// TIA Portal V19 export
FUNCTION "Route 406" : Void   // FC105, FBD
TITLE = Polygon Transfer Line - Production Sequence
{ S7_Optimized_Access := 'TRUE' }
// stored: AutoNumber false, SetENOAutomatically false
   VAR_TEMP
      device_fault : Bool;
      switch_fault : Bool;
      tmp : Bool;
      Step_on : Bool;
      Dev_Check : Bool;
      New_Msg : Bool;
      Route_Ready : Bool;   // Ready to Run
      PNIOnodeFault : Bool;
      StepTime : S5Time;
      TimerError : Int;
      scratch_DI : DInt;
      scratch_Real : Real;
      Message : Int;
      scratch_I : Int;
      tmpWord : Word;
      PNIODiag : Struct
         node_2 : Struct
            failed : Bool;
            moduleFault : Bool;
         END_STRUCT;
         node_3 : Struct
            failed : Bool;
            moduleFault : Bool;
         END_STRUCT;
         node_4 : Struct
            failed : Bool;
            moduleFault : Bool;
         END_STRUCT;
         node_5 : Struct
            failed : Bool;
            moduleFault : Bool;
         END_STRUCT;
         node_6 : Struct
            failed : Bool;
            moduleFault : Bool;
         END_STRUCT;
         node_7 : Struct
            failed : Bool;
            moduleFault : Bool;
         END_STRUCT;
         node_8 : Struct
            failed : Bool;
            moduleFault : Bool;
         END_STRUCT;
         node_9 : Struct
            failed : Bool;
            moduleFault : Bool;
         END_STRUCT;
         node_10 : Struct
            failed : Bool;
            moduleFault : Bool;
         END_STRUCT;
         node_11 : Struct
            failed : Bool;
            moduleFault : Bool;
            node_10 : Struct
               failed : Bool;
               moduleFault : Bool;
            END_STRUCT;
         END_STRUCT;
         node_12 : Struct
            failed : Bool;
            moduleFault : Bool;
         END_STRUCT;
      END_STRUCT;
      TV_above_zero : Bool;
      TV_equal_zero : Bool;
      PNIO_FaultActive : Bool;
   END_VAR
   VAR_TEMP   // added for the SCL form of the ladder/FBD networks
      _w1 : Bool;
   END_VAR
BEGIN

NETWORK
TITLE = PNIO 100 Node Faults
// PNIO Node 2
// PNIO Node 2
      A     "Module Diagnostic Result"."2_AL1103".ErrorValue.%X1;
      =     #PNIODiag.node_2.failed;
      A     "Module Diagnostic Result"."2_AL1103".ErrorValue.%X2;
      =     #PNIODiag.node_2.moduleFault;
// PNIO Node 3
      A     "Module Diagnostic Result"."3_AL1307".ErrorValue.%X1;
      =     #PNIODiag.node_3.failed;
      A     "Module Diagnostic Result"."3_AL1307".ErrorValue.%X2;
      =     #PNIODiag.node_3.moduleFault;
// PNIO Node 4
      A     "Module Diagnostic Result"."4_AL1307".ErrorValue.%X1;
      =     #PNIODiag.node_4.failed;
      A     "Module Diagnostic Result"."4_AL1307".ErrorValue.%X2;
      =     #PNIODiag.node_4.moduleFault;
// PNIO Node 5
      A     "Module Diagnostic Result"."5_AL1307".ErrorValue.%X1;
      =     #PNIODiag.node_5.failed;
      A     "Module Diagnostic Result"."5_AL1307".ErrorValue.%X2;
      =     #PNIODiag.node_5.moduleFault;
// PNIO Node 6
      A     "Module Diagnostic Result"."6_AL1307".ErrorValue.%X1;
      =     #PNIODiag.node_6.failed;
      A     "Module Diagnostic Result"."6_AL1307".ErrorValue.%X2;
      =     #PNIODiag.node_6.moduleFault;
// PNIO Node 7
      A     "Module Diagnostic Result"."7_AL1307".ErrorValue.%X1;
      =     #PNIODiag.node_7.failed;
      A     "Module Diagnostic Result"."7_AL1307".ErrorValue.%X2;
      =     #PNIODiag.node_7.moduleFault;
// PNIO Node 8
      A     "Module Diagnostic Result"."8_Promag300".ErrorValue.%X1;
      =     #PNIODiag.node_8.failed;
      A     "Module Diagnostic Result"."8_Promag300".ErrorValue.%X2;
      =     #PNIODiag.node_8.moduleFault;
// PNIO Node 9
      A     "Module Diagnostic Result"."9_SinaG120".ErrorValue.%X1;
      =     #PNIODiag.node_9.failed;
      A     "Module Diagnostic Result"."9_SinaG120".ErrorValue.%X2;
      =     #PNIODiag.node_9.moduleFault;
// PNIO Node 10
      A     "Module Diagnostic Result"."10_AL1307".ErrorValue.%X1;
      =     #PNIODiag.node_10.failed;
      A     "Module Diagnostic Result"."10_AL1307".ErrorValue.%X2;
      =     #PNIODiag.node_10.moduleFault;
// PNIO Node 11
      A     "Module Diagnostic Result"."11_PNCoup".ErrorValue.%X1;
      =     #PNIODiag.node_11.failed;
      A     "Module Diagnostic Result"."11_PNCoup".ErrorValue.%X2;
      =     #PNIODiag.node_11.moduleFault;
// PNIO Node 12
      A     "Module Diagnostic Result"."12_AL1307".ErrorValue.%X1;
      =     #PNIODiag.node_12.failed;
      A     "Module Diagnostic Result"."12_AL1307".ErrorValue.%X2;
      =     #PNIODiag.node_12.moduleFault;


NETWORK
TITLE = PNIO node fault
      O     #PNIODiag.node_2.failed;
      O     #PNIODiag.node_2.moduleFault;
      O     #PNIODiag.node_3.failed;
      O     #PNIODiag.node_3.moduleFault;
      O     #PNIODiag.node_4.failed;
      O     #PNIODiag.node_4.moduleFault;
      O     #PNIODiag.node_5.failed;
      O     #PNIODiag.node_5.moduleFault;
      O     #PNIODiag.node_6.failed;
      O     #PNIODiag.node_6.moduleFault;
      O     #PNIODiag.node_7.failed;
      O     #PNIODiag.node_7.moduleFault;
      O     #PNIODiag.node_8.failed;
      O     #PNIODiag.node_8.moduleFault;
      O     #PNIODiag.node_9.failed;
      O     #PNIODiag.node_9.moduleFault;
      O     #PNIODiag.node_10.failed;
      O     #PNIODiag.node_10.moduleFault;
      O     #PNIODiag.node_11.failed;
      O     #PNIODiag.node_11.moduleFault;
      O     #PNIODiag.node_12.failed;
      O     #PNIODiag.node_12.moduleFault;
      AN    "RTE_406_DB".HMI_CMD.PNIO_FaultOverride;
      =     #PNIOnodeFault;


NETWORK
TITLE = PNIO Override
      A     "RTE_406_DB".HMI.SEQUENCE_HELD;
      A     #PNIOnodeFault;
      AN(;
      L     "IO-LinkDevicesDB".AL2221_100_005_X06.DeviceStatus;
      L     0;
      >I;
      O     #PNIODiag.node_5.failed;
      );
      S     "RTE_406_DB".HMI_CMD.PNIO_FaultOverrideAvail;

      AN    "RTE_406_DB".HMI.RUNNING;
      R     "RTE_406_DB".HMI_CMD.PNIO_FaultOverrideAvail;
      R     "RTE_406_DB".HMI_CMD.PNIO_FaultOverride;

REGION Network 4: Device Faults
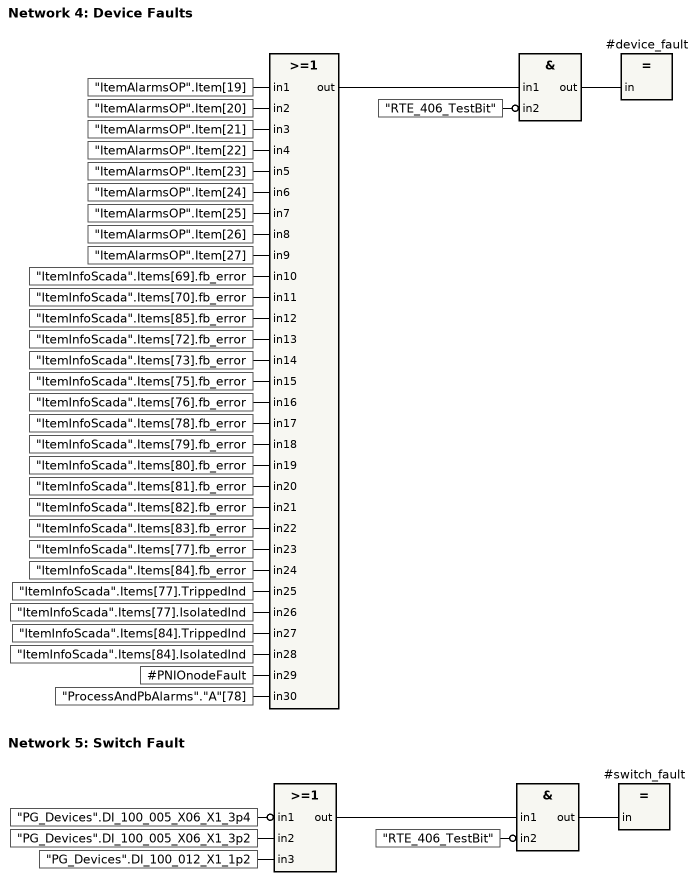
   #device_fault := ("ItemAlarmsOP".Item[19] OR "ItemAlarmsOP".Item[20] OR "ItemAlarmsOP".Item[21] OR "ItemAlarmsOP".Item[22] OR "ItemAlarmsOP".Item[23] OR "ItemAlarmsOP".Item[24] OR "ItemAlarmsOP".Item[25] OR "ItemAlarmsOP".Item[26] OR "ItemAlarmsOP".Item[27] OR "ItemInfoScada".Items[69].fb_error OR "ItemInfoScada".Items[70].fb_error OR "ItemInfoScada".Items[85].fb_error OR "ItemInfoScada".Items[72].fb_error OR "ItemInfoScada".Items[73].fb_error OR "ItemInfoScada".Items[75].fb_error OR "ItemInfoScada".Items[76].fb_error OR "ItemInfoScada".Items[78].fb_error OR "ItemInfoScada".Items[79].fb_error OR "ItemInfoScada".Items[80].fb_error OR "ItemInfoScada".Items[81].fb_error OR "ItemInfoScada".Items[82].fb_error OR "ItemInfoScada".Items[83].fb_error OR "ItemInfoScada".Items[77].fb_error OR "ItemInfoScada".Items[84].fb_error OR "ItemInfoScada".Items[77].TrippedInd OR "ItemInfoScada".Items[77].IsolatedInd OR "ItemInfoScada".Items[84].TrippedInd OR "ItemInfoScada".Items[84].IsolatedInd OR #PNIOnodeFault OR "ProcessAndPbAlarms"."A"[78]) AND NOT "RTE_406_TestBit";
END_REGION

REGION Network 5: Switch Fault
   #switch_fault := (NOT "PG_Devices".DI_100_005_X06_X1_3p4 OR "PG_Devices".DI_100_005_X06_X1_3p2 OR "PG_Devices".DI_100_012_X1_1p2) AND NOT "RTE_406_TestBit";
END_REGION

REGION Network 6: Set Devices in Auto
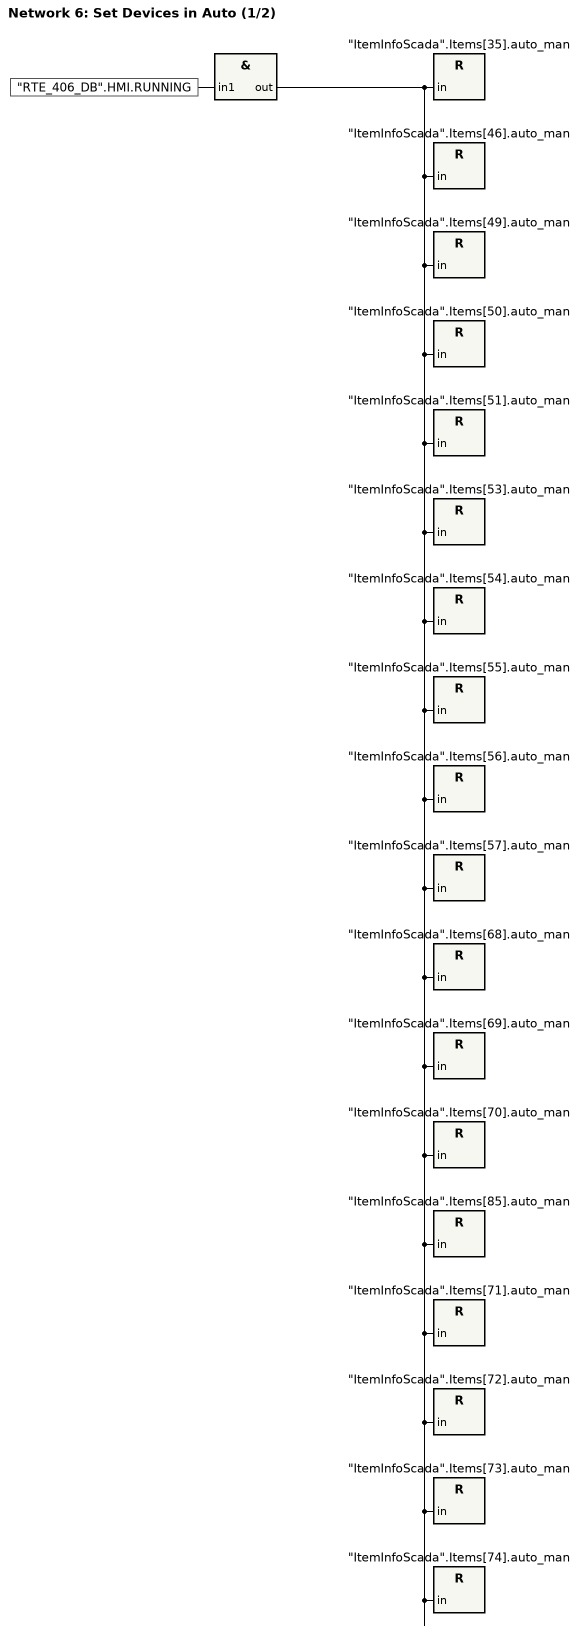
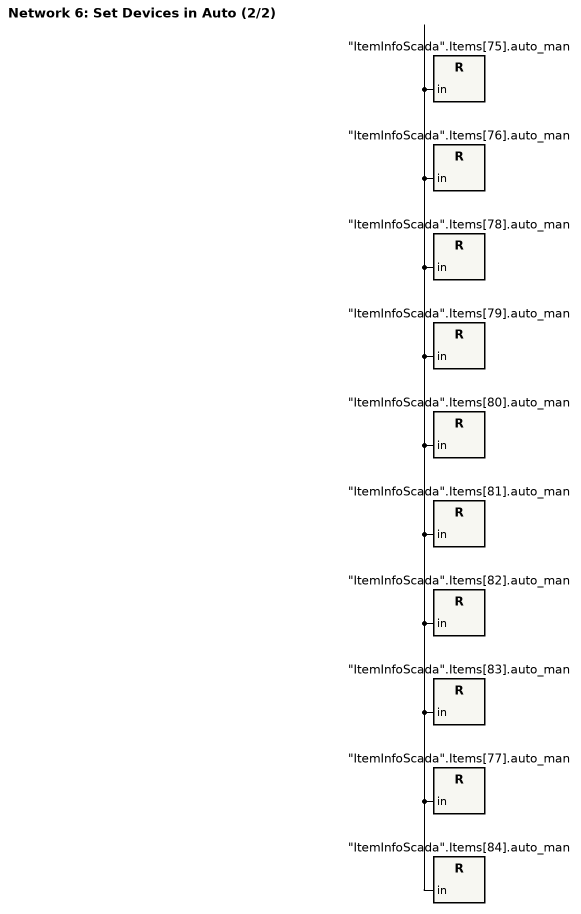
   IF "RTE_406_DB".HMI.RUNNING THEN
       "ItemInfoScada".Items[35].auto_man := FALSE;
       "ItemInfoScada".Items[46].auto_man := FALSE;
       "ItemInfoScada".Items[49].auto_man := FALSE;
       "ItemInfoScada".Items[50].auto_man := FALSE;
       "ItemInfoScada".Items[51].auto_man := FALSE;
       "ItemInfoScada".Items[53].auto_man := FALSE;
       "ItemInfoScada".Items[54].auto_man := FALSE;
       "ItemInfoScada".Items[55].auto_man := FALSE;
       "ItemInfoScada".Items[56].auto_man := FALSE;
       "ItemInfoScada".Items[57].auto_man := FALSE;
       "ItemInfoScada".Items[68].auto_man := FALSE;
       "ItemInfoScada".Items[69].auto_man := FALSE;
       "ItemInfoScada".Items[70].auto_man := FALSE;
       "ItemInfoScada".Items[85].auto_man := FALSE;
       "ItemInfoScada".Items[71].auto_man := FALSE;
       "ItemInfoScada".Items[72].auto_man := FALSE;
       "ItemInfoScada".Items[73].auto_man := FALSE;
       "ItemInfoScada".Items[74].auto_man := FALSE;
       "ItemInfoScada".Items[75].auto_man := FALSE;
       "ItemInfoScada".Items[76].auto_man := FALSE;
       "ItemInfoScada".Items[78].auto_man := FALSE;
       "ItemInfoScada".Items[79].auto_man := FALSE;
       "ItemInfoScada".Items[80].auto_man := FALSE;
       "ItemInfoScada".Items[81].auto_man := FALSE;
       "ItemInfoScada".Items[82].auto_man := FALSE;
       "ItemInfoScada".Items[83].auto_man := FALSE;
       "ItemInfoScada".Items[77].auto_man := FALSE;
       "ItemInfoScada".Items[84].auto_man := FALSE;
   END_IF;
END_REGION

REGION Network 7: Route Healthy
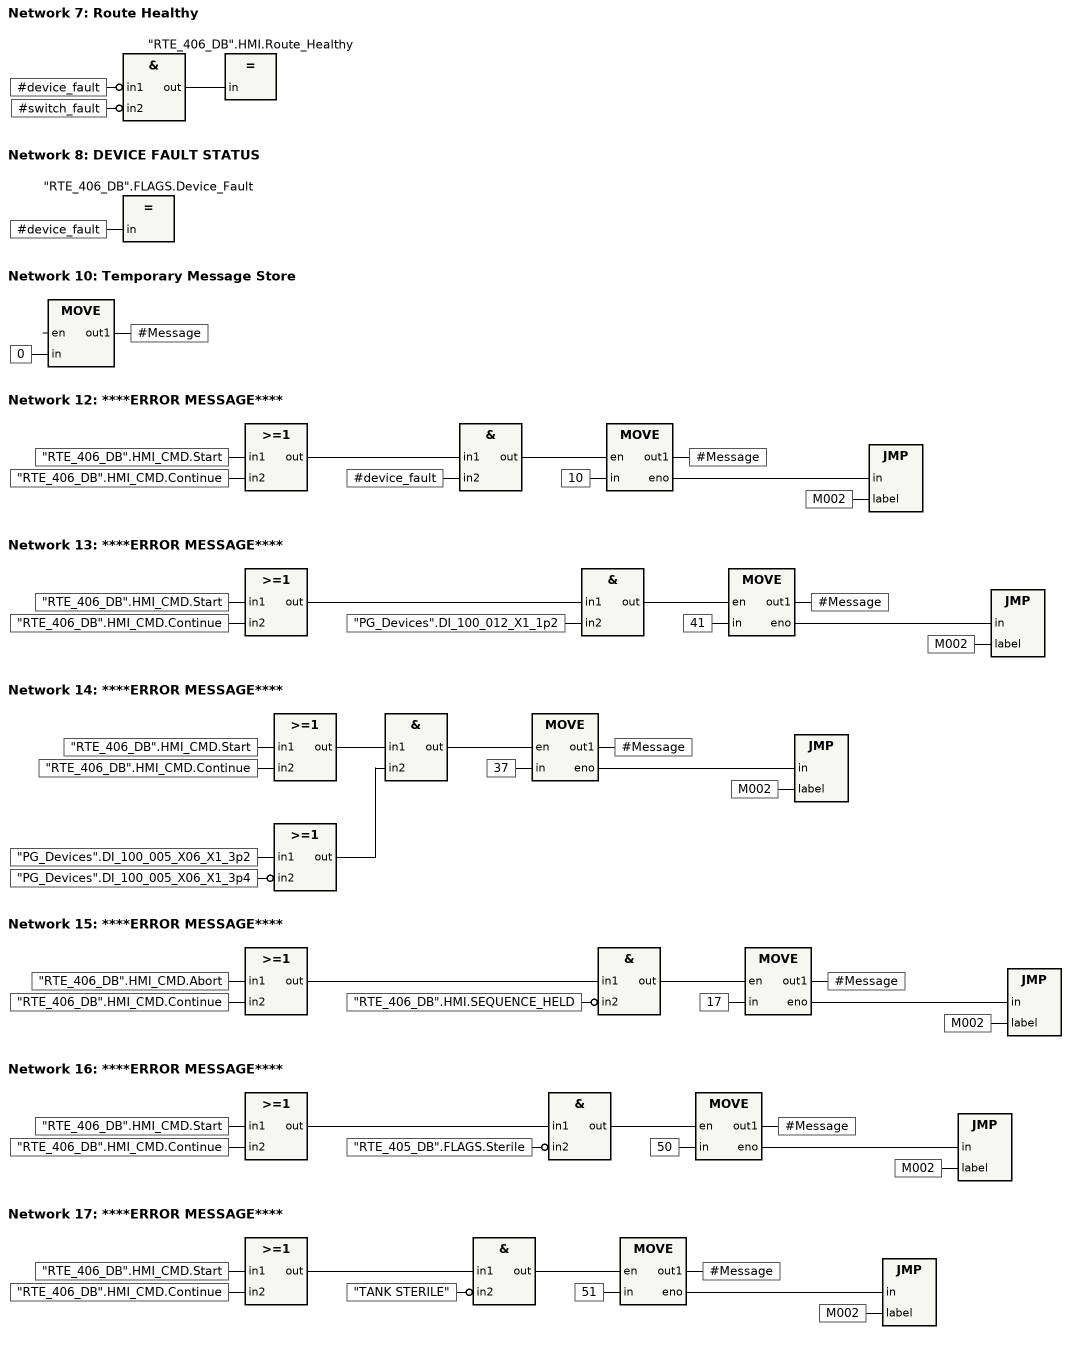
   "RTE_406_DB".HMI.Route_Healthy := NOT #device_fault AND NOT #switch_fault;
END_REGION

REGION Network 8: DEVICE FAULT STATUS
   "RTE_406_DB".FLAGS.Device_Fault := #device_fault;
END_REGION

NETWORK
TITLE = GENERAL FAULT STATUS
      O     #switch_fault;
      O     "RTE_406_DB".FLAGS.Device_Fault;
      A     "RTE_406_DB".HMI.RUNNING;
      =     "RTE_406_DB".HMI.FAULT;

REGION Network 10: Temporary Message Store
   // Clear down temporary message store.
   #Message := 0;
END_REGION

NETWORK
TITLE = Generate Sequence Start Command
// The sequence is initiated via the interface signals ..afl
      A     "RTE_406_DB".HMI_CMD.Start;
      AN    "RTE_406_DB".HMI.RUNNING;
      A     "RTE_406_DB".HMI.Route_Healthy;
      =     "RTE_406_DB".FLAGS.Sequence_Start;

      AN    "RTE_406_DB".HMI.RUNNING;
      A     "RTE_406_DB".HMI.Route_Healthy;
      =     "RTE_406_DB".HMI_CMD.Start_Available;


REGION Network 12: ****ERROR MESSAGE****
   // Message 10 - Device Fault
   // ENO of a box is taken as its EN; it also drops when the box reports an error
   #_w1 := ("RTE_406_DB".HMI_CMD.Start OR "RTE_406_DB".HMI_CMD.Continue) AND #device_fault;
   IF #_w1 THEN
       #Message := 10;
       GOTO M002;
   END_IF;
END_REGION

REGION Network 13: ****ERROR MESSAGE****
   // Message 41 - Forward Control Stop activated
   // ENO of a box is taken as its EN; it also drops when the box reports an error
   #_w1 := ("RTE_406_DB".HMI_CMD.Start OR "RTE_406_DB".HMI_CMD.Continue) AND "PG_Devices".DI_100_012_X1_1p2;
   IF #_w1 THEN
       #Message := 41;
       GOTO M002;
   END_IF;
END_REGION

REGION Network 14: ****ERROR MESSAGE****
   // Message 37 - Swingbend out of position
   // ENO of a box is taken as its EN; it also drops when the box reports an error
   #_w1 := ("RTE_406_DB".HMI_CMD.Start OR "RTE_406_DB".HMI_CMD.Continue) AND ("PG_Devices".DI_100_005_X06_X1_3p2 OR NOT "PG_Devices".DI_100_005_X06_X1_3p4);
   IF #_w1 THEN
       #Message := 37;
       GOTO M002;
   END_IF;
END_REGION

REGION Network 15: ****ERROR MESSAGE****
   // Message 17 - Sequence Not Held
   // To abort or continue the clean it must have already been held.
   // ENO of a box is taken as its EN; it also drops when the box reports an error
   #_w1 := ("RTE_406_DB".HMI_CMD.Abort OR "RTE_406_DB".HMI_CMD.Continue) AND NOT "RTE_406_DB".HMI.SEQUENCE_HELD;
   IF #_w1 THEN
       #Message := 17;
       GOTO M002;
   END_IF;
END_REGION

REGION Network 16: ****ERROR MESSAGE****
   // Message 50 - Line not Sterile
   // ENO of a box is taken as its EN; it also drops when the box reports an error
   #_w1 := ("RTE_406_DB".HMI_CMD.Start OR "RTE_406_DB".HMI_CMD.Continue) AND NOT "RTE_405_DB".FLAGS.Sterile;
   IF #_w1 THEN
       #Message := 50;
       GOTO M002;
   END_IF;
END_REGION

REGION Network 17: ****ERROR MESSAGE****
   // Message 51 - AHV Not Sterile
   // ENO of a box is taken as its EN; it also drops when the box reports an error
   #_w1 := ("RTE_406_DB".HMI_CMD.Start OR "RTE_406_DB".HMI_CMD.Continue) AND NOT "TANK STERILE";
   IF #_w1 THEN
       #Message := 51;
       GOTO M002;
   END_IF;
END_REGION

REGION Network 18: ****ERROR MESSAGE****
   // Message 28 - Filler Not Sterile
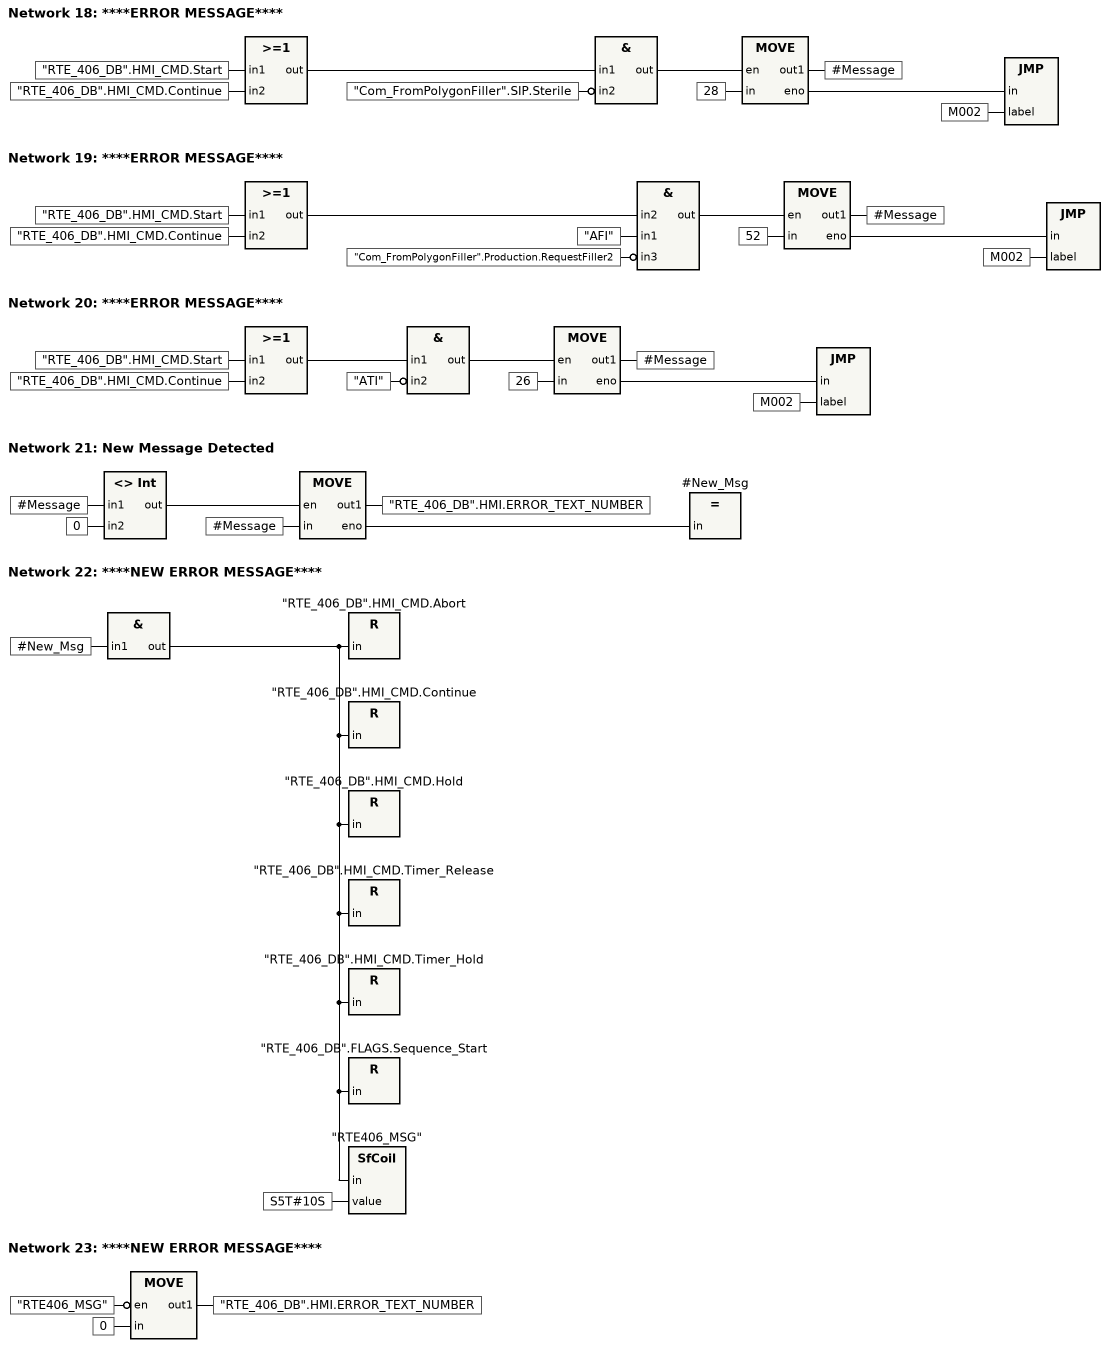
   // ENO of a box is taken as its EN; it also drops when the box reports an error
   #_w1 := ("RTE_406_DB".HMI_CMD.Start OR "RTE_406_DB".HMI_CMD.Continue) AND NOT "Com_FromPolygonFiller".SIP.Sterile;
   IF #_w1 THEN
       #Message := 28;
       GOTO M002;
   END_IF;
END_REGION

REGION Network 19: ****ERROR MESSAGE****
   // Message 52 - No Product Request From Filler
   // ENO of a box is taken as its EN; it also drops when the box reports an error
   #_w1 := ("RTE_406_DB".HMI_CMD.Start OR "RTE_406_DB".HMI_CMD.Continue) AND "AFI" AND NOT "Com_FromPolygonFiller".Production.RequestFiller2;
   IF #_w1 THEN
       #Message := 52;
       GOTO M002;
   END_IF;
END_REGION

REGION Network 20: ****ERROR MESSAGE****
   // Message xx - Tank low level for production start
   // Check text msg number
   // ENO of a box is taken as its EN; it also drops when the box reports an error
   #_w1 := ("RTE_406_DB".HMI_CMD.Start OR "RTE_406_DB".HMI_CMD.Continue) AND NOT "ATI";
   IF #_w1 THEN
       #Message := 26;
       GOTO M002;
   END_IF;
END_REGION

REGION Network 21: New Message Detected
   // ENO of a box is taken as its EN; it also drops when the box reports an error
   M002:
   #_w1 := #Message <> 0;
   IF #_w1 THEN "RTE_406_DB".HMI.ERROR_TEXT_NUMBER := #Message; END_IF;
   #New_Msg := #_w1;
END_REGION

REGION Network 22: ****NEW ERROR MESSAGE****
   // Reset all CIP commands except START.
   // On a new non-zero error message being displayed reset all commands from SCADA 
   // so they take no action. Also, start a delay off timer to cancel display of the 
   // error message.
   // no SCL statement known for SfCoil: written as a call
   IF #New_Msg THEN
       "RTE_406_DB".HMI_CMD.Abort := FALSE;
       "RTE_406_DB".HMI_CMD.Continue := FALSE;
       "RTE_406_DB".HMI_CMD.Hold := FALSE;
       "RTE_406_DB".HMI_CMD.Timer_Release := FALSE;
       "RTE_406_DB".HMI_CMD.Timer_Hold := FALSE;
       "RTE_406_DB".FLAGS.Sequence_Start := FALSE;
   END_IF;
   SfCoil(in := #New_Msg, value := S5T#10S, operand := "RTE406_MSG");
END_REGION

REGION Network 23: ****NEW ERROR MESSAGE****
   // Error message display cancel.
   IF NOT "RTE406_MSG" THEN "RTE_406_DB".HMI.ERROR_TEXT_NUMBER := 0; END_IF;
END_REGION

REGION Network 24: ROUTE RUNNING
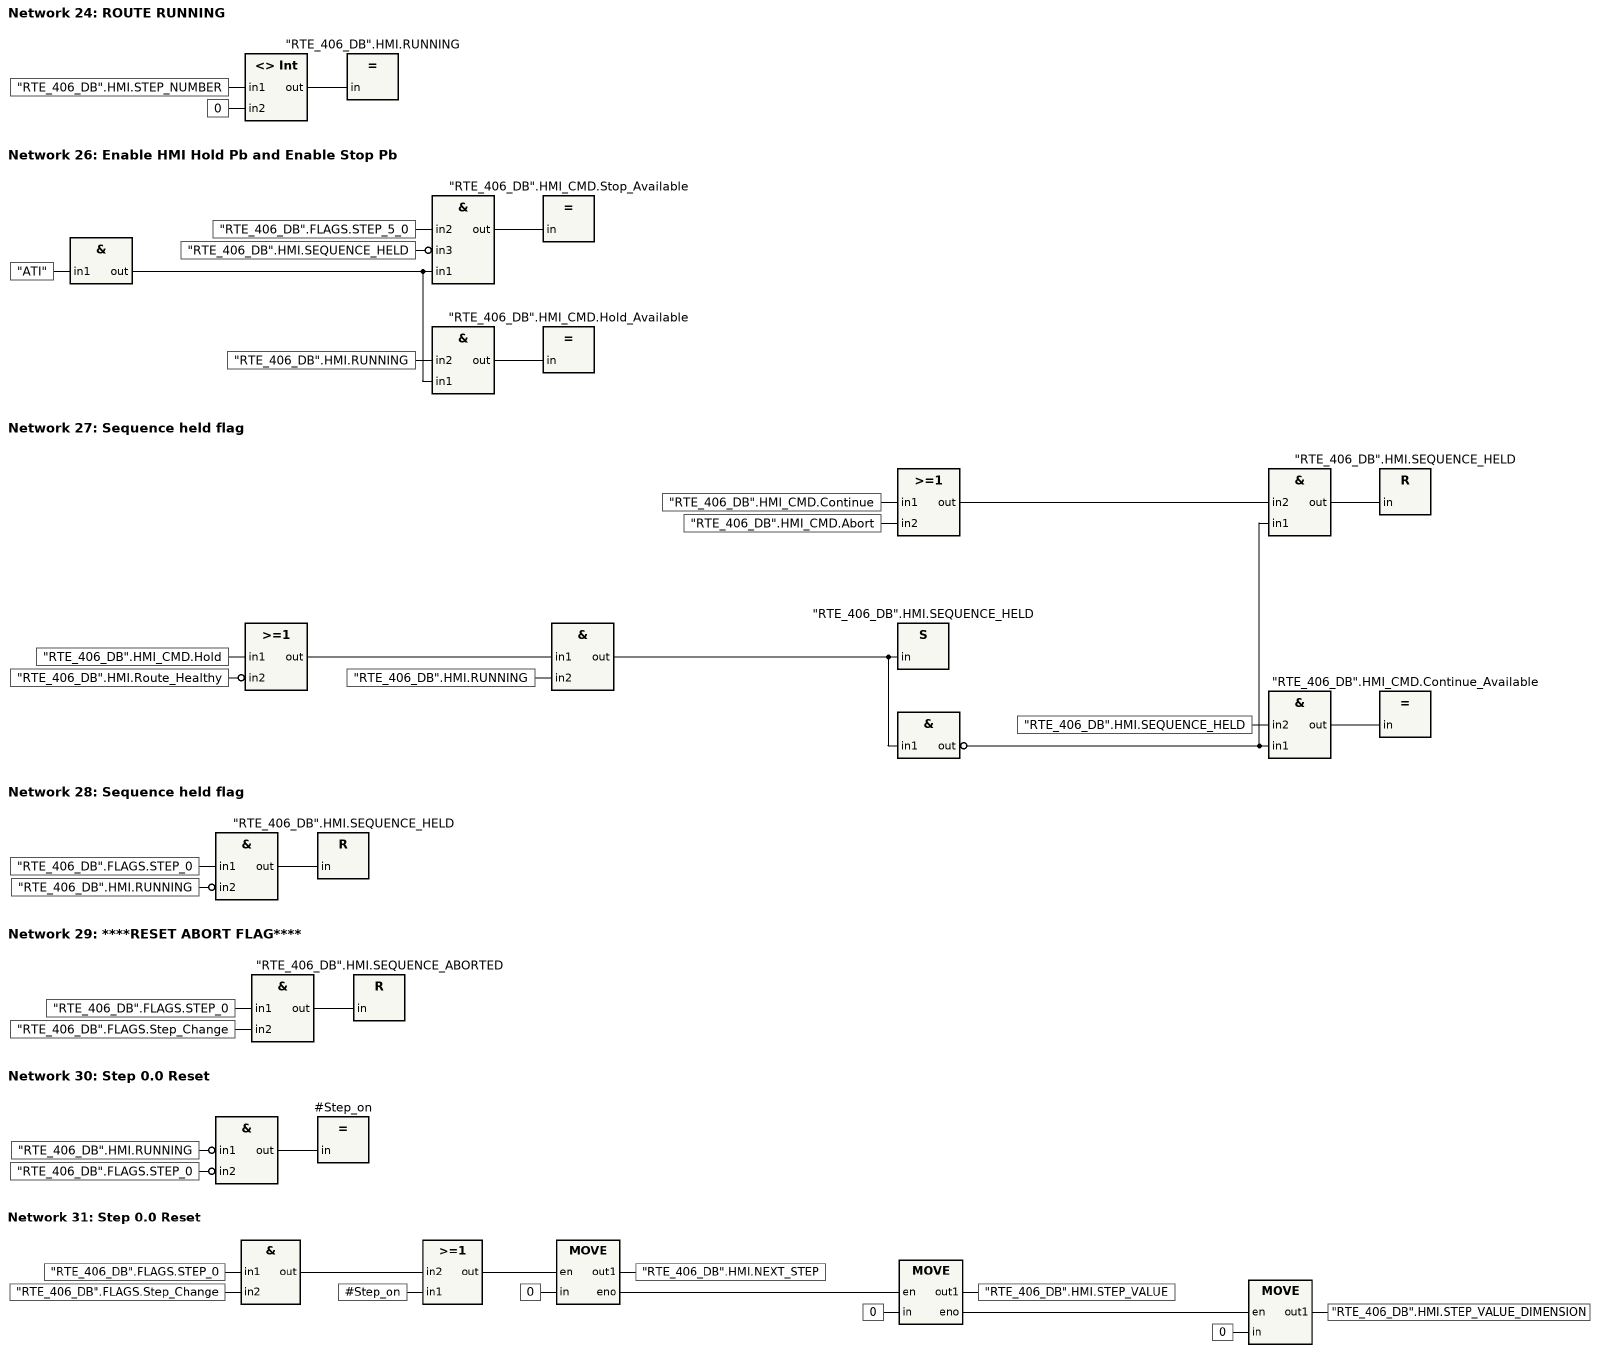
   "RTE_406_DB".HMI.RUNNING := "RTE_406_DB".HMI.STEP_NUMBER <> 0;
END_REGION

NETWORK
TITLE = ****SEQ ABORT****
      A     "RTE_406_DB".HMI_CMD.Abort;
      A     "RTE_406_DB".HMI.SEQUENCE_HELD;
      S     "RTE_406_DB".HMI.SEQUENCE_ABORTED;

      A     "RTE_406_DB".HMI.SEQUENCE_HELD;
      =     "RTE_406_DB".HMI_CMD.Abort_Available;

REGION Network 26: Enable HMI Hold Pb and Enable Stop Pb
   "RTE_406_DB".HMI_CMD.Hold_Available := "RTE_406_DB".HMI.RUNNING AND "ATI";
   "RTE_406_DB".HMI_CMD.Stop_Available := "RTE_406_DB".FLAGS.STEP_5_0 AND NOT "RTE_406_DB".HMI.SEQUENCE_HELD AND "ATI";
END_REGION

REGION Network 27: Sequence held flag
   // Set sequence hold if sequence is running and a hold fault condition is detected 
   // or a sequence hold command is received from SCADA.
   // 
   // When a validated CONTINUE command is received from SCADA and all fault 
   // conditions are cleared then reset sequence hold.
   #_w1 := ("RTE_406_DB".HMI_CMD.Hold OR NOT "RTE_406_DB".HMI.Route_Healthy) AND "RTE_406_DB".HMI.RUNNING;
   IF #_w1 THEN "RTE_406_DB".HMI.SEQUENCE_HELD := TRUE; END_IF;
   IF ("RTE_406_DB".HMI_CMD.Continue OR "RTE_406_DB".HMI_CMD.Abort) AND NOT #_w1 THEN
       "RTE_406_DB".HMI.SEQUENCE_HELD := FALSE;
   END_IF;
   "RTE_406_DB".HMI_CMD.Continue_Available := "RTE_406_DB".HMI.SEQUENCE_HELD AND NOT #_w1;
END_REGION

REGION Network 28: Sequence held flag
   // Reset when circuit not running i.e after an abort.
   IF "RTE_406_DB".FLAGS.STEP_0 AND NOT "RTE_406_DB".HMI.RUNNING THEN
       "RTE_406_DB".HMI.SEQUENCE_HELD := FALSE;
   END_IF;
END_REGION

REGION Network 29: ****RESET ABORT FLAG****
   IF "RTE_406_DB".FLAGS.STEP_0 AND "RTE_406_DB".FLAGS.Step_Change THEN
       "RTE_406_DB".HMI.SEQUENCE_ABORTED := FALSE;
   END_IF;
END_REGION

REGION Network 30: Step 0.0 Reset
   #Step_on := NOT "RTE_406_DB".HMI.RUNNING AND NOT "RTE_406_DB".FLAGS.STEP_0;
END_REGION

REGION Network 31: Step 0.0 Reset
   // Reset sequnece to step 0 and clear down step value and dimension words.
   // ENO of a box is taken as its EN; it also drops when the box reports an error
   IF ("RTE_406_DB".FLAGS.STEP_0 AND "RTE_406_DB".FLAGS.Step_Change) OR #Step_on THEN
       "RTE_406_DB".HMI.NEXT_STEP := 0;
       "RTE_406_DB".HMI.STEP_VALUE := 0;
       "RTE_406_DB".HMI.STEP_VALUE_DIMENSION := 0;
   END_IF;
END_REGION

REGION Network 32: Move to Step 0.5
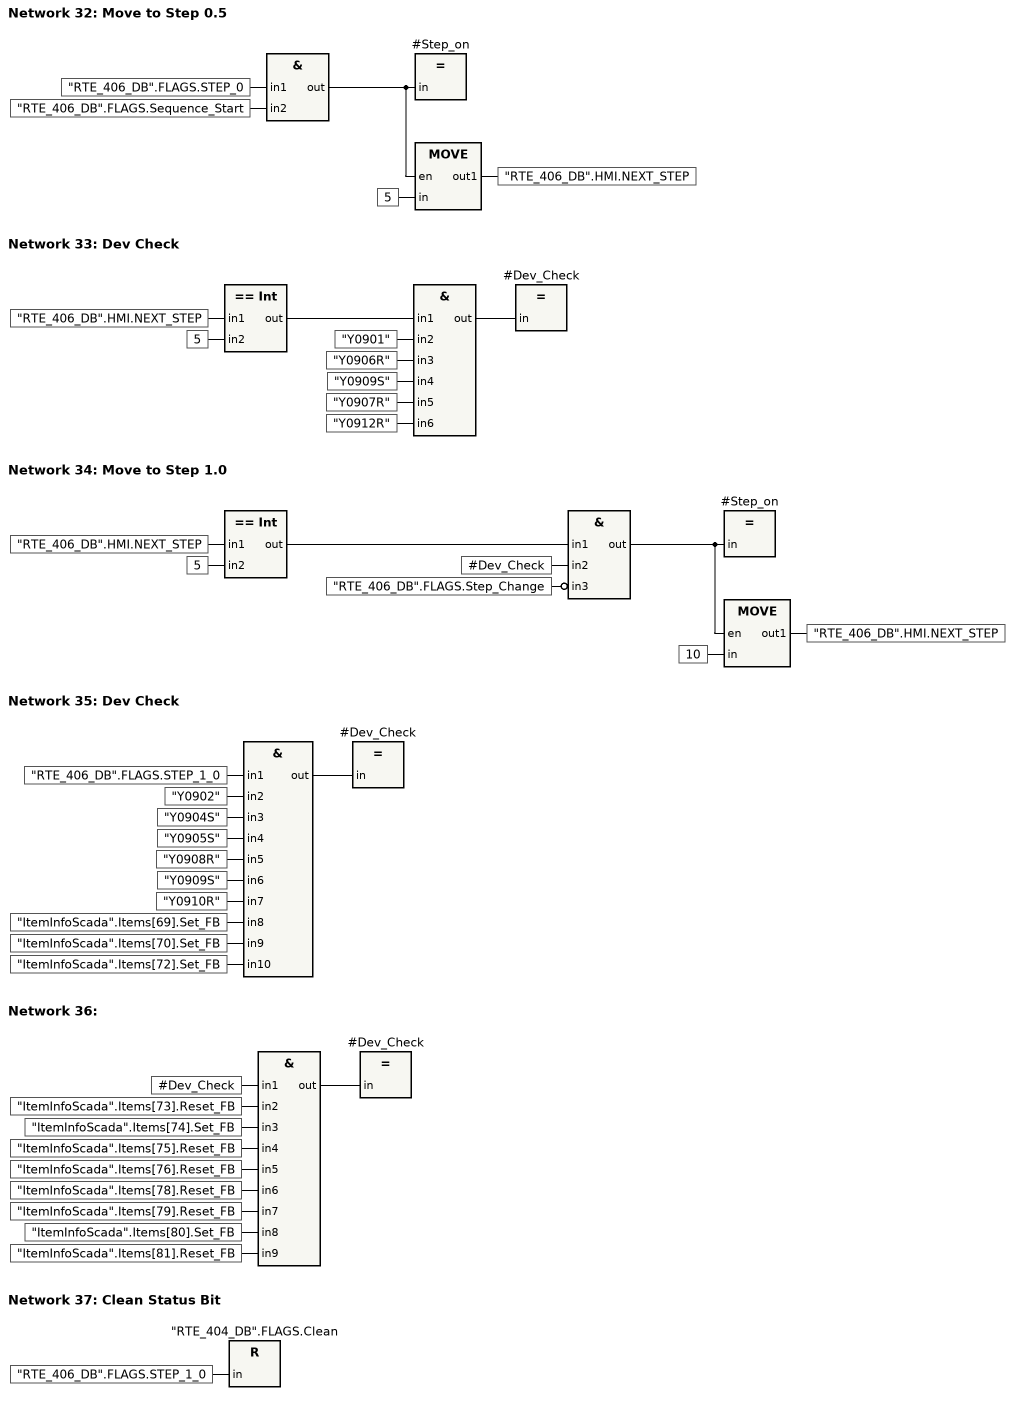
   #Step_on := "RTE_406_DB".FLAGS.STEP_0 AND "RTE_406_DB".FLAGS.Sequence_Start;
   IF #Step_on THEN "RTE_406_DB".HMI.NEXT_STEP := 5; END_IF;
END_REGION

REGION Network 33: Dev Check
   // Dev Check following Route valves Open - 09.10, 09.08, 09.45, 10.21, 10.23, 10.25
   // and following Route Valves closed - 09.09, 09.05, 10.24
   #Dev_Check := ("RTE_406_DB".HMI.NEXT_STEP = 5) AND "Y0901" AND "Y0906R" AND "Y0909S" AND "Y0907R" AND "Y0912R";
END_REGION

REGION Network 34: Move to Step 1.0
   #Step_on := ("RTE_406_DB".HMI.NEXT_STEP = 5) AND #Dev_Check AND NOT "RTE_406_DB".FLAGS.Step_Change;
   IF #Step_on THEN "RTE_406_DB".HMI.NEXT_STEP := 10; END_IF;
END_REGION

REGION Network 35: Dev Check
   // Dev Check following Route valves Open - 09.10, 09.08, 09.45, 10.21, 10.23, 10.25
   // and following Route Valves closed - 09.09, 09.05, 10.24
   #Dev_Check := "RTE_406_DB".FLAGS.STEP_1_0 AND "Y0902" AND "Y0904S" AND "Y0905S" AND "Y0908R" AND "Y0909S" AND "Y0910R" AND "ItemInfoScada".Items[69].Set_FB AND "ItemInfoScada".Items[70].Set_FB AND "ItemInfoScada".Items[72].Set_FB;
END_REGION

REGION Network 36
   #Dev_Check := #Dev_Check AND "ItemInfoScada".Items[73].Reset_FB AND "ItemInfoScada".Items[74].Set_FB AND "ItemInfoScada".Items[75].Reset_FB AND "ItemInfoScada".Items[76].Reset_FB AND "ItemInfoScada".Items[78].Reset_FB AND "ItemInfoScada".Items[79].Reset_FB AND "ItemInfoScada".Items[80].Set_FB AND "ItemInfoScada".Items[81].Reset_FB;
END_REGION

REGION Network 37: Clean Status Bit
   IF "RTE_406_DB".FLAGS.STEP_1_0 THEN "RTE_404_DB".FLAGS.Clean := FALSE; END_IF;
END_REGION

REGION Network 38: Move to Step 2.0
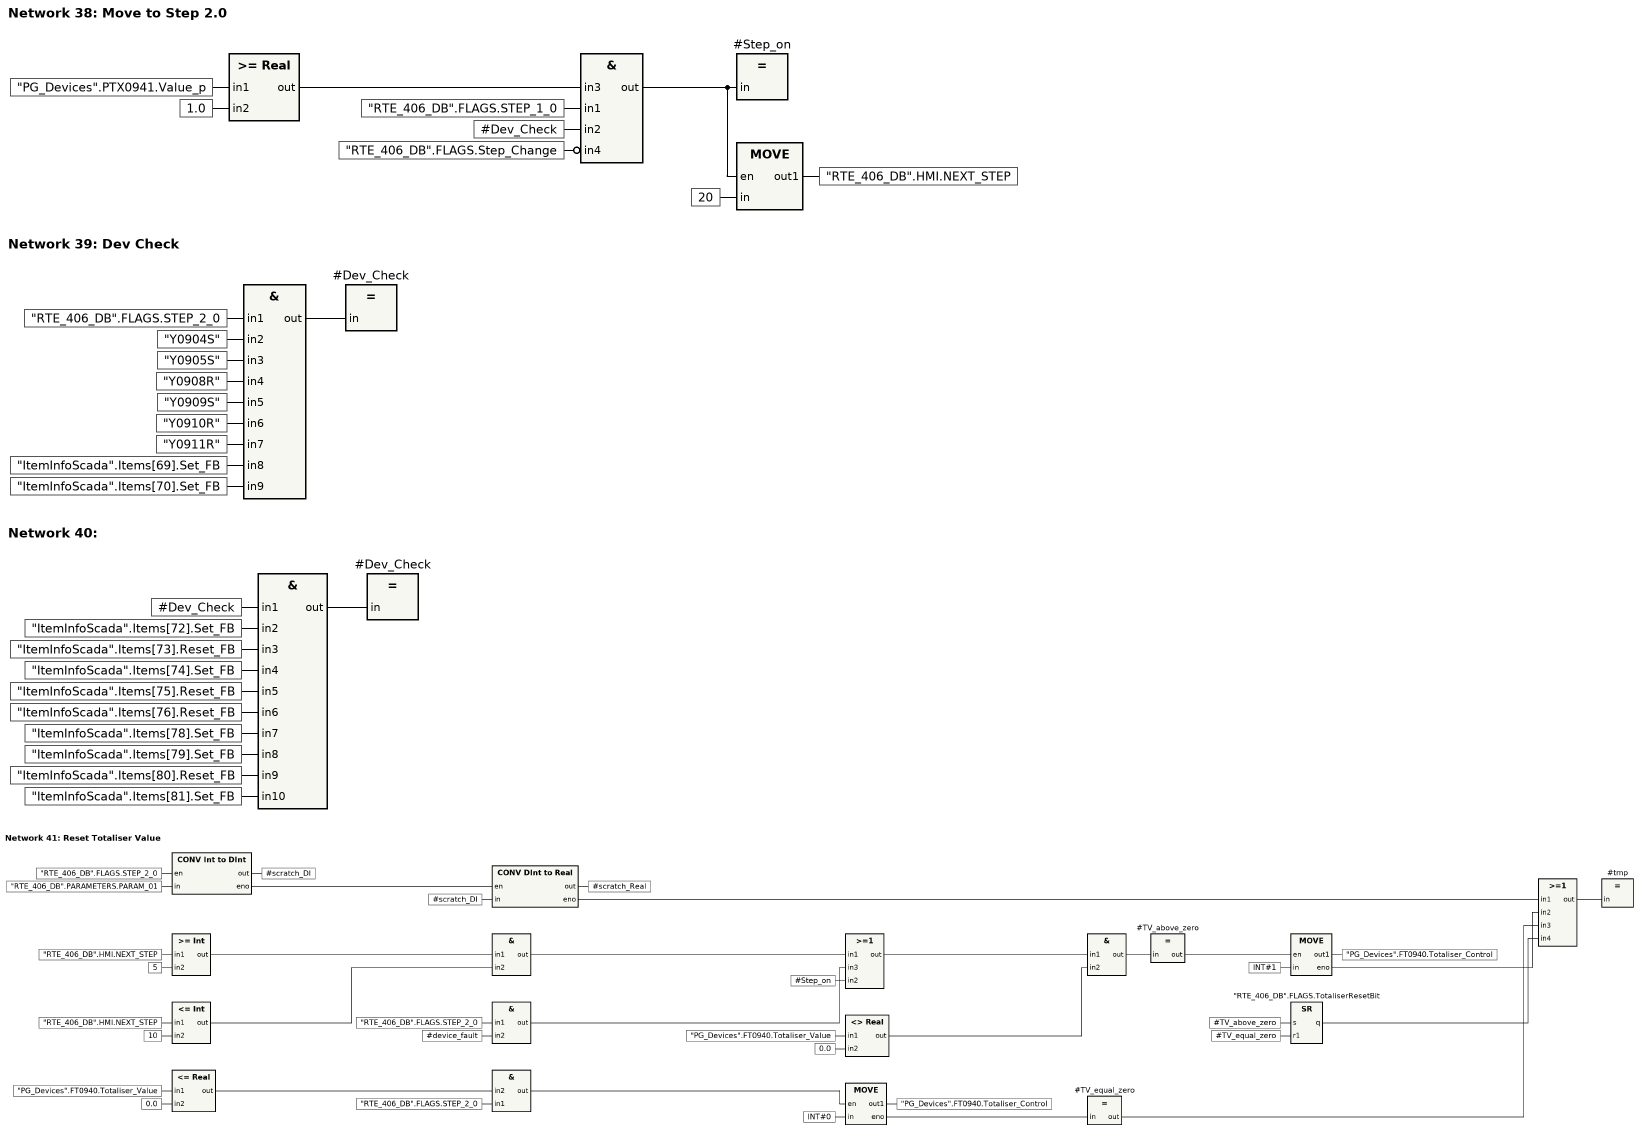
   #Step_on := ("PG_Devices".PTX0941.Value_p >= 1.0) AND "RTE_406_DB".FLAGS.STEP_1_0 AND #Dev_Check AND NOT "RTE_406_DB".FLAGS.Step_Change;
   IF #Step_on THEN "RTE_406_DB".HMI.NEXT_STEP := 20; END_IF;
END_REGION

REGION Network 39: Dev Check
   // Dev Check following Route valves Open - 09.10, 09.08, 09.45, 10.21, 10.23, 10.25
   // and following Route Valves closed - 09.09, 09.05, 10.24
   #Dev_Check := "RTE_406_DB".FLAGS.STEP_2_0 AND "Y0904S" AND "Y0905S" AND "Y0908R" AND "Y0909S" AND "Y0910R" AND "Y0911R" AND "ItemInfoScada".Items[69].Set_FB AND "ItemInfoScada".Items[70].Set_FB;
END_REGION

REGION Network 40
   #Dev_Check := #Dev_Check AND "ItemInfoScada".Items[72].Set_FB AND "ItemInfoScada".Items[73].Reset_FB AND "ItemInfoScada".Items[74].Set_FB AND "ItemInfoScada".Items[75].Reset_FB AND "ItemInfoScada".Items[76].Reset_FB AND "ItemInfoScada".Items[78].Set_FB AND "ItemInfoScada".Items[79].Set_FB AND "ItemInfoScada".Items[80].Reset_FB AND "ItemInfoScada".Items[81].Set_FB;
END_REGION

REGION Network 41: Reset Totaliser Value
   // Totaliser Control
   // 0 = Totalise
   // 3 = Reset + Totalise
   // ENO of a box is taken as its EN; it also drops when the box reports an error
   IF "RTE_406_DB".FLAGS.STEP_2_0 THEN
       #scratch_DI := INT_TO_DINT("RTE_406_DB".PARAMETERS.PARAM_01);
       #scratch_Real := DINT_TO_REAL(#scratch_DI);
   END_IF;
   #TV_above_zero := ((("RTE_406_DB".HMI.NEXT_STEP >= 5) AND ("RTE_406_DB".HMI.NEXT_STEP <= 10)) OR ("RTE_406_DB".FLAGS.STEP_2_0 AND #device_fault) OR #Step_on) AND ("PG_Devices".FT0940.Totaliser_Value <> 0.0);
   IF #TV_above_zero THEN "PG_Devices".FT0940.Totaliser_Control := INT#1; END_IF;
   #_w1 := ("PG_Devices".FT0940.Totaliser_Value <= 0.0) AND "RTE_406_DB".FLAGS.STEP_2_0;
   IF #_w1 THEN "PG_Devices".FT0940.Totaliser_Control := INT#0; END_IF;
   #TV_equal_zero := #_w1;
   IF #TV_above_zero THEN
       "RTE_406_DB".FLAGS.TotaliserResetBit := TRUE;   // SR flip-flop
   END_IF;
   IF #TV_equal_zero THEN "RTE_406_DB".FLAGS.TotaliserResetBit := FALSE; END_IF;
   #tmp := "RTE_406_DB".FLAGS.STEP_2_0 OR #TV_above_zero OR #_w1 OR "RTE_406_DB".FLAGS.TotaliserResetBit;
END_REGION

REGION Network 42: Move to Step 3.0
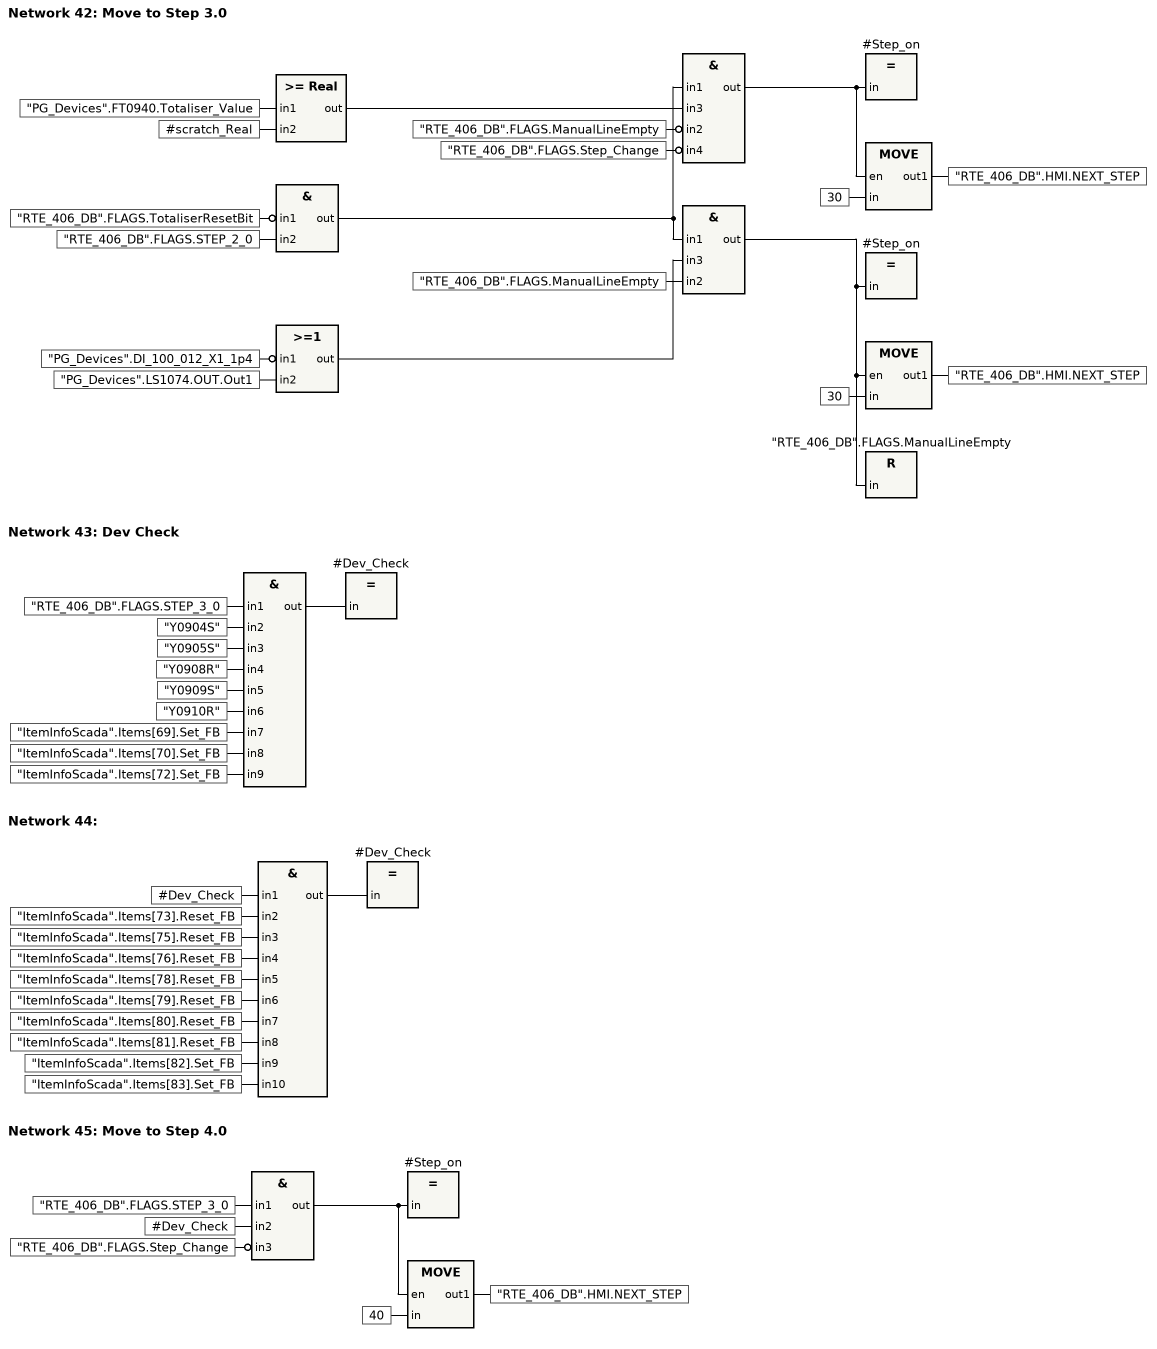
   #_w1 := NOT "RTE_406_DB".FLAGS.TotaliserResetBit AND "RTE_406_DB".FLAGS.STEP_2_0;
   #Step_on := #_w1 AND ("PG_Devices".FT0940.Totaliser_Value >= #scratch_Real) AND NOT "RTE_406_DB".FLAGS.ManualLineEmpty AND NOT "RTE_406_DB".FLAGS.Step_Change;
   IF #Step_on THEN "RTE_406_DB".HMI.NEXT_STEP := 30; END_IF;
   #Step_on := #_w1 AND (NOT "PG_Devices".DI_100_012_X1_1p4 OR "PG_Devices".LS1074.OUT.Out1) AND "RTE_406_DB".FLAGS.ManualLineEmpty;
   IF #Step_on THEN
       "RTE_406_DB".HMI.NEXT_STEP := 30;
       "RTE_406_DB".FLAGS.ManualLineEmpty := FALSE;
   END_IF;
END_REGION

REGION Network 43: Dev Check
   // Dev Check following Route valves Open - 09.10, 09.08, 09.45, 10.21, 10.23, 10.25
   // and following Route Valves closed - 09.09, 09.05, 10.24
   #Dev_Check := "RTE_406_DB".FLAGS.STEP_3_0 AND "Y0904S" AND "Y0905S" AND "Y0908R" AND "Y0909S" AND "Y0910R" AND "ItemInfoScada".Items[69].Set_FB AND "ItemInfoScada".Items[70].Set_FB AND "ItemInfoScada".Items[72].Set_FB;
END_REGION

REGION Network 44
   #Dev_Check := #Dev_Check AND "ItemInfoScada".Items[73].Reset_FB AND "ItemInfoScada".Items[75].Reset_FB AND "ItemInfoScada".Items[76].Reset_FB AND "ItemInfoScada".Items[78].Reset_FB AND "ItemInfoScada".Items[79].Reset_FB AND "ItemInfoScada".Items[80].Reset_FB AND "ItemInfoScada".Items[81].Reset_FB AND "ItemInfoScada".Items[82].Set_FB AND "ItemInfoScada".Items[83].Set_FB;
END_REGION

REGION Network 45: Move to Step 4.0
   #Step_on := "RTE_406_DB".FLAGS.STEP_3_0 AND #Dev_Check AND NOT "RTE_406_DB".FLAGS.Step_Change;
   IF #Step_on THEN "RTE_406_DB".HMI.NEXT_STEP := 40; END_IF;
END_REGION

REGION Network 46: Initialise Step Parameters
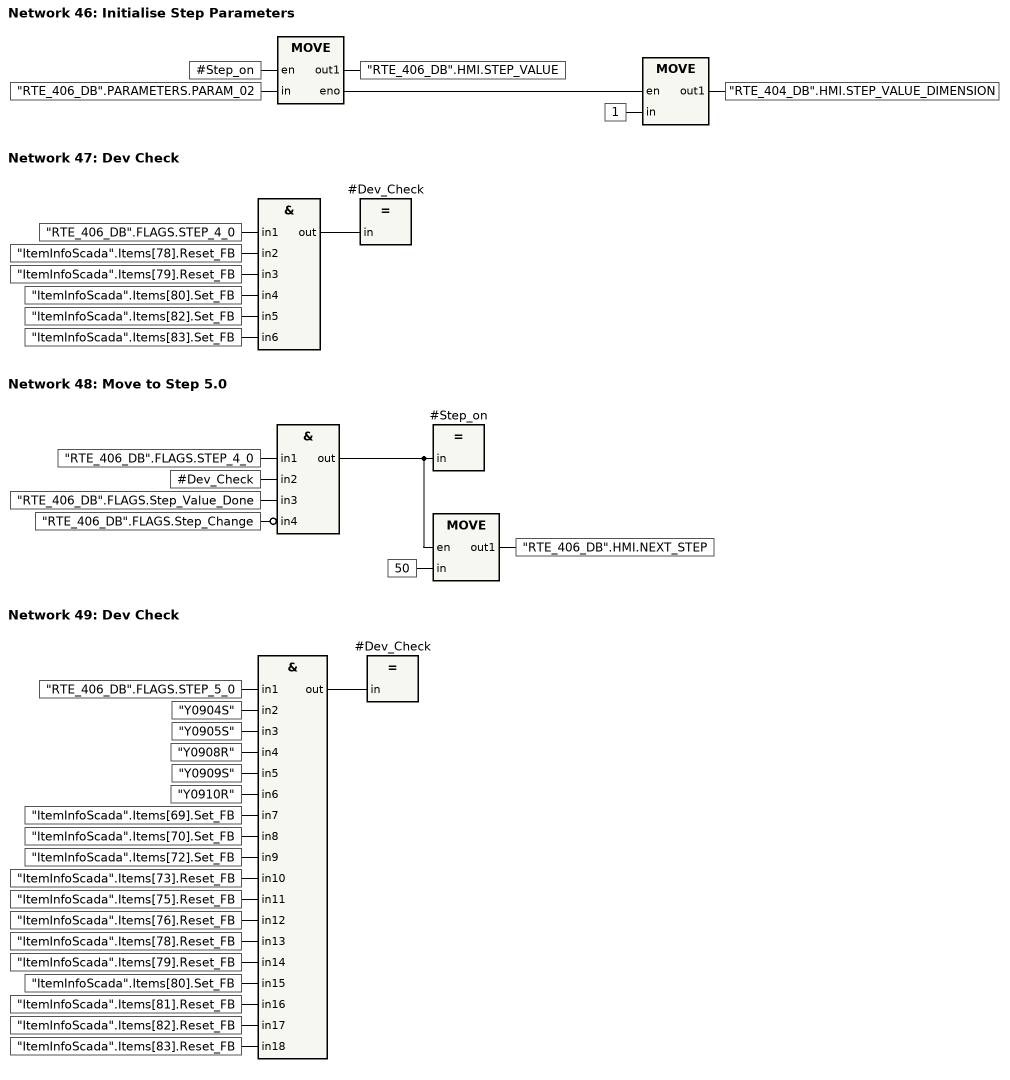
   // ENO of a box is taken as its EN; it also drops when the box reports an error
   IF #Step_on THEN
       "RTE_406_DB".HMI.STEP_VALUE := "RTE_406_DB".PARAMETERS.PARAM_02;
       "RTE_404_DB".HMI.STEP_VALUE_DIMENSION := 1;
   END_IF;
END_REGION

REGION Network 47: Dev Check
   // Dev Check following Route valves Open - 09.10, 09.08, 09.45, 10.21, 10.23, 10.25
   // and following Route Valves closed - 09.09, 09.05, 10.24
   #Dev_Check := "RTE_406_DB".FLAGS.STEP_4_0 AND "ItemInfoScada".Items[78].Reset_FB AND "ItemInfoScada".Items[79].Reset_FB AND "ItemInfoScada".Items[80].Set_FB AND "ItemInfoScada".Items[82].Set_FB AND "ItemInfoScada".Items[83].Set_FB;
END_REGION

REGION Network 48: Move to Step 5.0
   #Step_on := "RTE_406_DB".FLAGS.STEP_4_0 AND #Dev_Check AND "RTE_406_DB".FLAGS.Step_Value_Done AND NOT "RTE_406_DB".FLAGS.Step_Change;
   IF #Step_on THEN "RTE_406_DB".HMI.NEXT_STEP := 50; END_IF;
END_REGION

REGION Network 49: Dev Check
   // Dev Check following Route valves Open - 09.10, 09.08, 09.45, 10.21, 10.23, 10.25
   // and following Route Valves closed - 09.09, 09.05, 10.24
   #Dev_Check := "RTE_406_DB".FLAGS.STEP_5_0 AND "Y0904S" AND "Y0905S" AND "Y0908R" AND "Y0909S" AND "Y0910R" AND "ItemInfoScada".Items[69].Set_FB AND "ItemInfoScada".Items[70].Set_FB AND "ItemInfoScada".Items[72].Set_FB AND "ItemInfoScada".Items[73].Reset_FB AND "ItemInfoScada".Items[75].Reset_FB AND "ItemInfoScada".Items[76].Reset_FB AND "ItemInfoScada".Items[78].Reset_FB AND "ItemInfoScada".Items[79].Reset_FB AND "ItemInfoScada".Items[80].Set_FB AND "ItemInfoScada".Items[81].Reset_FB AND "ItemInfoScada".Items[82].Reset_FB AND "ItemInfoScada".Items[83].Reset_FB;
END_REGION

REGION Network 50: Move to Step 6.0
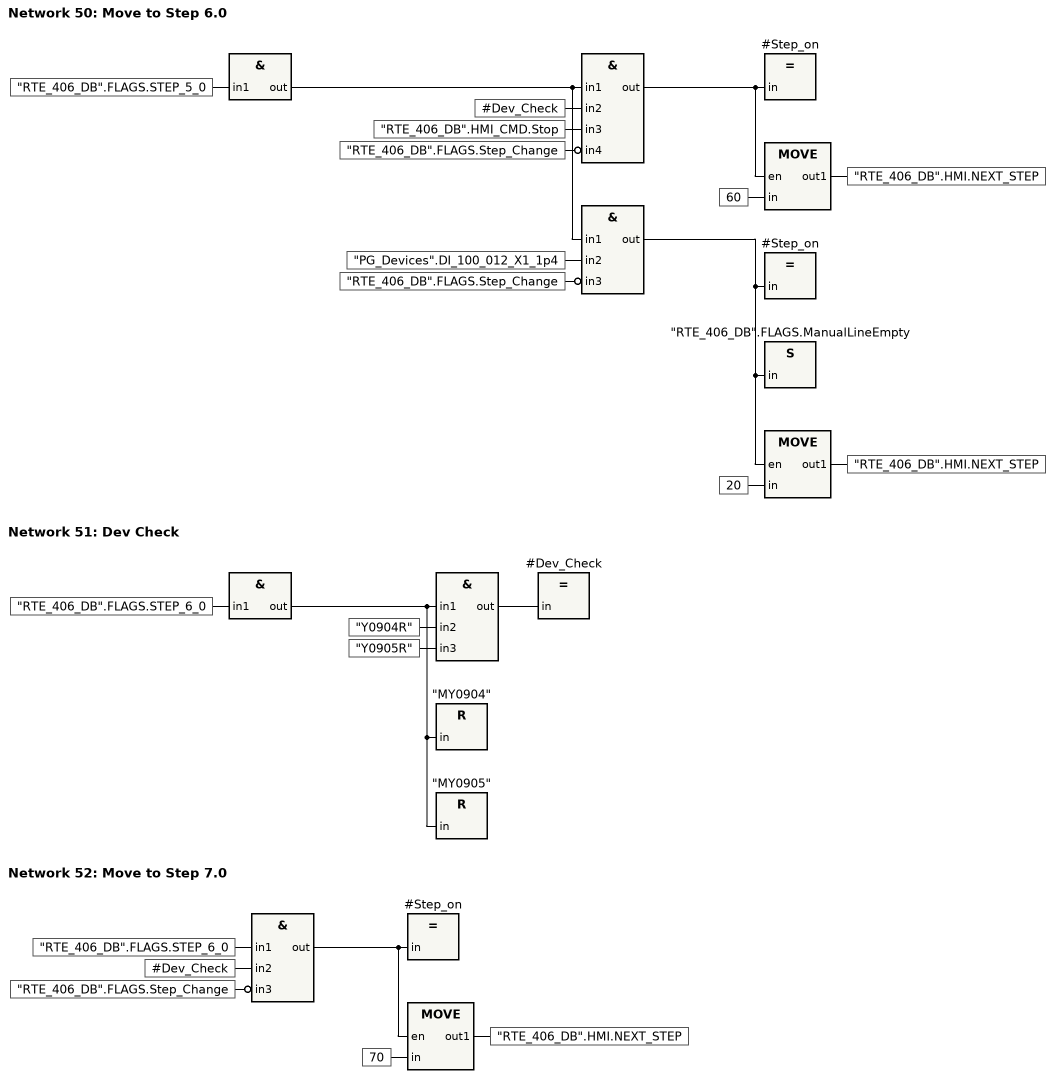
   #Step_on := "RTE_406_DB".FLAGS.STEP_5_0 AND #Dev_Check AND "RTE_406_DB".HMI_CMD.Stop AND NOT "RTE_406_DB".FLAGS.Step_Change;
   IF #Step_on THEN "RTE_406_DB".HMI.NEXT_STEP := 60; END_IF;
   #Step_on := "RTE_406_DB".FLAGS.STEP_5_0 AND "PG_Devices".DI_100_012_X1_1p4 AND NOT "RTE_406_DB".FLAGS.Step_Change;
   IF #Step_on THEN
       "RTE_406_DB".FLAGS.ManualLineEmpty := TRUE;
       "RTE_406_DB".HMI.NEXT_STEP := 20;
   END_IF;
END_REGION

REGION Network 51: Dev Check
   // Dev Check following Route valves Open - 09.10, 09.08, 09.45, 10.21, 10.23, 10.25
   // and following Route Valves closed - 09.09, 09.05, 10.24
   #Dev_Check := "RTE_406_DB".FLAGS.STEP_6_0 AND "Y0904R" AND "Y0905R";
   IF "RTE_406_DB".FLAGS.STEP_6_0 THEN
       "MY0904" := FALSE;
       "MY0905" := FALSE;
   END_IF;
END_REGION

REGION Network 52: Move to Step 7.0
   #Step_on := "RTE_406_DB".FLAGS.STEP_6_0 AND #Dev_Check AND NOT "RTE_406_DB".FLAGS.Step_Change;
   IF #Step_on THEN "RTE_406_DB".HMI.NEXT_STEP := 70; END_IF;
END_REGION

REGION Network 53: Dev Check
   // Dev Check following Route valves Open - 09.10, 09.08, 09.45, 10.21, 10.23, 10.25
   // and following Route Valves closed - 09.09, 09.05, 10.24
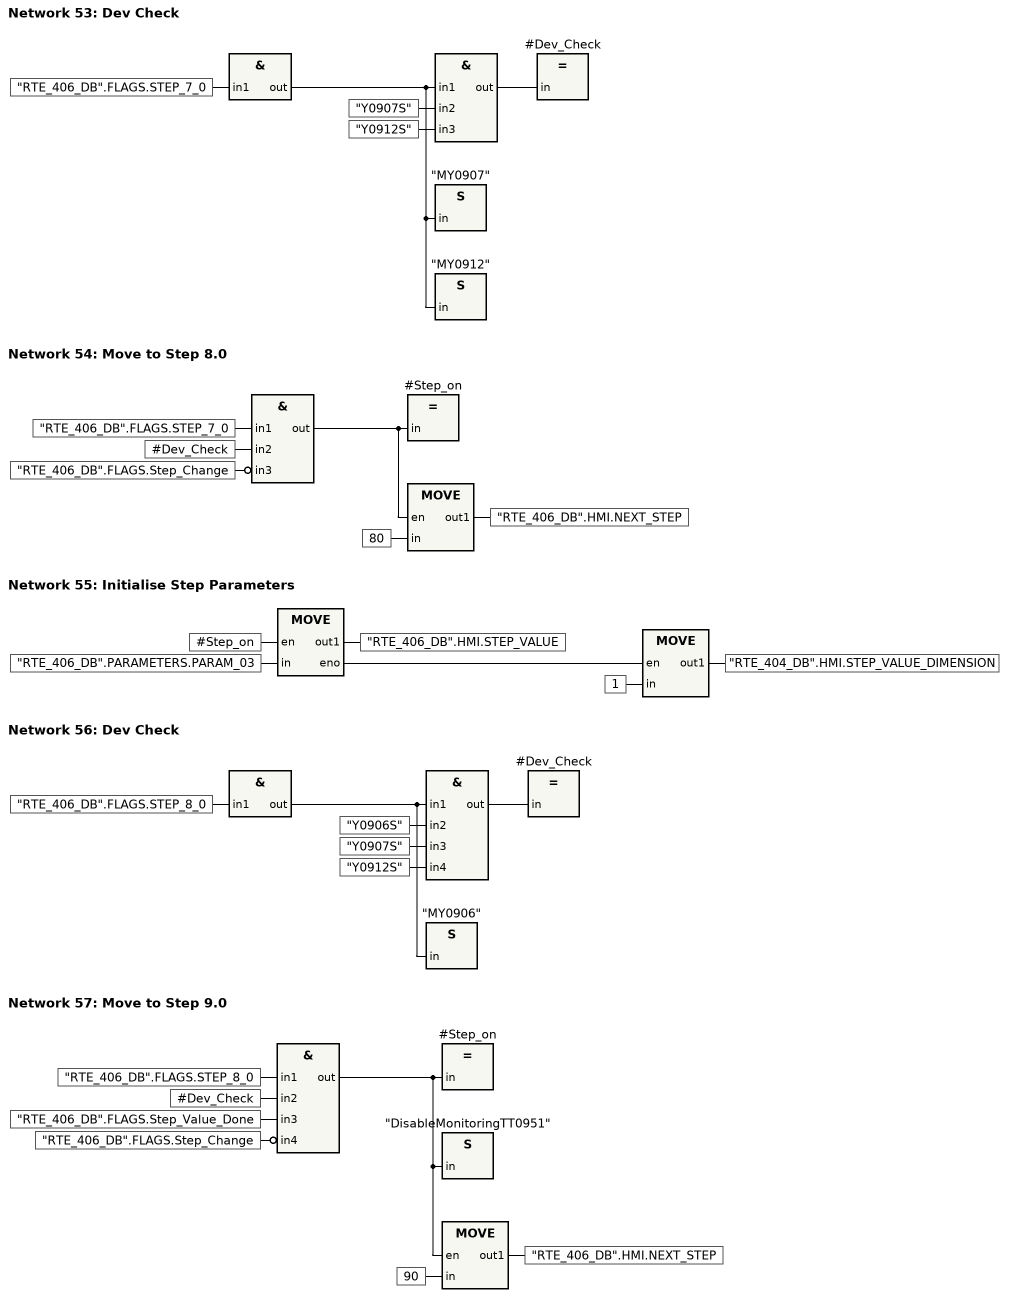
   #Dev_Check := "RTE_406_DB".FLAGS.STEP_7_0 AND "Y0907S" AND "Y0912S";
   IF "RTE_406_DB".FLAGS.STEP_7_0 THEN
       "MY0907" := TRUE;
       "MY0912" := TRUE;
   END_IF;
END_REGION

REGION Network 54: Move to Step 8.0
   #Step_on := "RTE_406_DB".FLAGS.STEP_7_0 AND #Dev_Check AND NOT "RTE_406_DB".FLAGS.Step_Change;
   IF #Step_on THEN "RTE_406_DB".HMI.NEXT_STEP := 80; END_IF;
END_REGION

REGION Network 55: Initialise Step Parameters
   // ENO of a box is taken as its EN; it also drops when the box reports an error
   IF #Step_on THEN
       "RTE_406_DB".HMI.STEP_VALUE := "RTE_406_DB".PARAMETERS.PARAM_03;
       "RTE_404_DB".HMI.STEP_VALUE_DIMENSION := 1;
   END_IF;
END_REGION

REGION Network 56: Dev Check
   // Dev Check 
   // ** Disable TT0951 monitoring
   #Dev_Check := "RTE_406_DB".FLAGS.STEP_8_0 AND "Y0906S" AND "Y0907S" AND "Y0912S";
   IF "RTE_406_DB".FLAGS.STEP_8_0 THEN "MY0906" := TRUE; END_IF;
END_REGION

REGION Network 57: Move to Step 9.0
   #Step_on := "RTE_406_DB".FLAGS.STEP_8_0 AND #Dev_Check AND "RTE_406_DB".FLAGS.Step_Value_Done AND NOT "RTE_406_DB".FLAGS.Step_Change;
   IF #Step_on THEN
       "DisableMonitoringTT0951" := TRUE;
       "RTE_406_DB".HMI.NEXT_STEP := 90;
   END_IF;
END_REGION

REGION Network 58: Dev Check
   // Dev Check 
   // ** Enable TT0951 monitoring
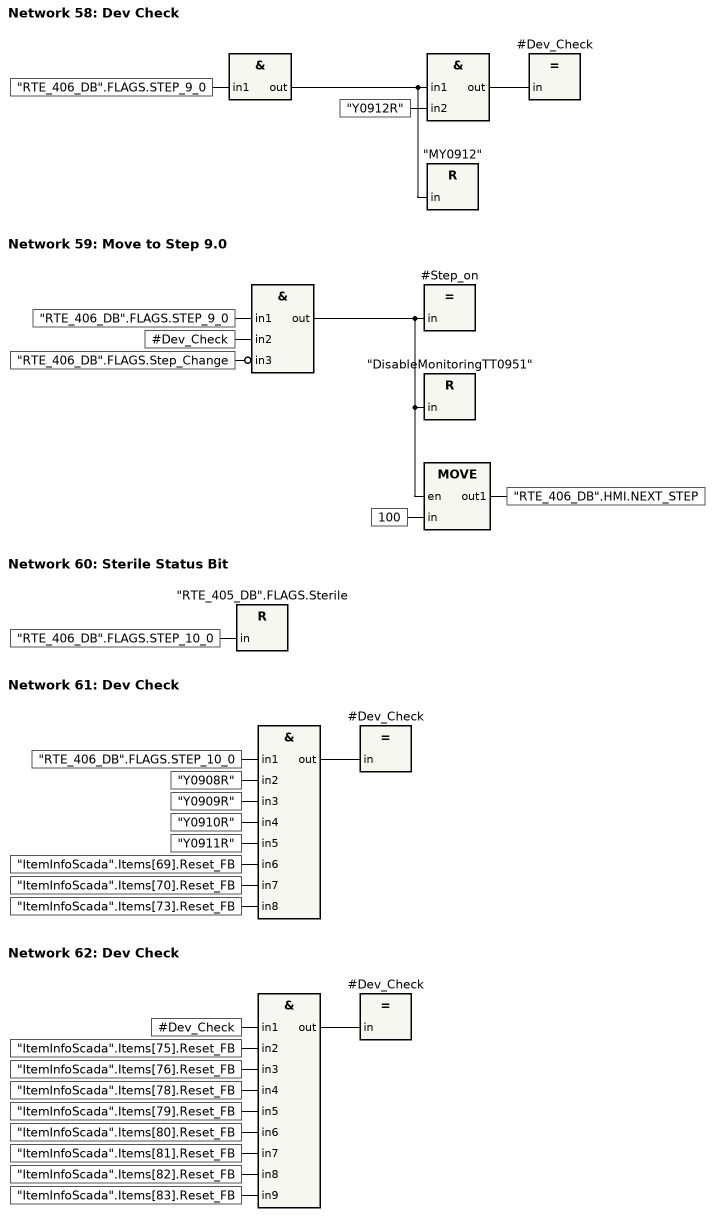
   #Dev_Check := "RTE_406_DB".FLAGS.STEP_9_0 AND "Y0912R";
   IF "RTE_406_DB".FLAGS.STEP_9_0 THEN "MY0912" := FALSE; END_IF;
END_REGION

REGION Network 59: Move to Step 9.0
   #Step_on := "RTE_406_DB".FLAGS.STEP_9_0 AND #Dev_Check AND NOT "RTE_406_DB".FLAGS.Step_Change;
   IF #Step_on THEN
       "DisableMonitoringTT0951" := FALSE;
       "RTE_406_DB".HMI.NEXT_STEP := 100;
   END_IF;
END_REGION

REGION Network 60: Sterile Status Bit
   IF "RTE_406_DB".FLAGS.STEP_10_0 THEN "RTE_405_DB".FLAGS.Sterile := FALSE; END_IF;
END_REGION

REGION Network 61: Dev Check
   // Dev Check
   #Dev_Check := "RTE_406_DB".FLAGS.STEP_10_0 AND "Y0908R" AND "Y0909R" AND "Y0910R" AND "Y0911R" AND "ItemInfoScada".Items[69].Reset_FB AND "ItemInfoScada".Items[70].Reset_FB AND "ItemInfoScada".Items[73].Reset_FB;
END_REGION

REGION Network 62: Dev Check
   // Dev Check
   #Dev_Check := #Dev_Check AND "ItemInfoScada".Items[75].Reset_FB AND "ItemInfoScada".Items[76].Reset_FB AND "ItemInfoScada".Items[78].Reset_FB AND "ItemInfoScada".Items[79].Reset_FB AND "ItemInfoScada".Items[80].Reset_FB AND "ItemInfoScada".Items[81].Reset_FB AND "ItemInfoScada".Items[82].Reset_FB AND "ItemInfoScada".Items[83].Reset_FB;
END_REGION

REGION Network 63: Move to Step End
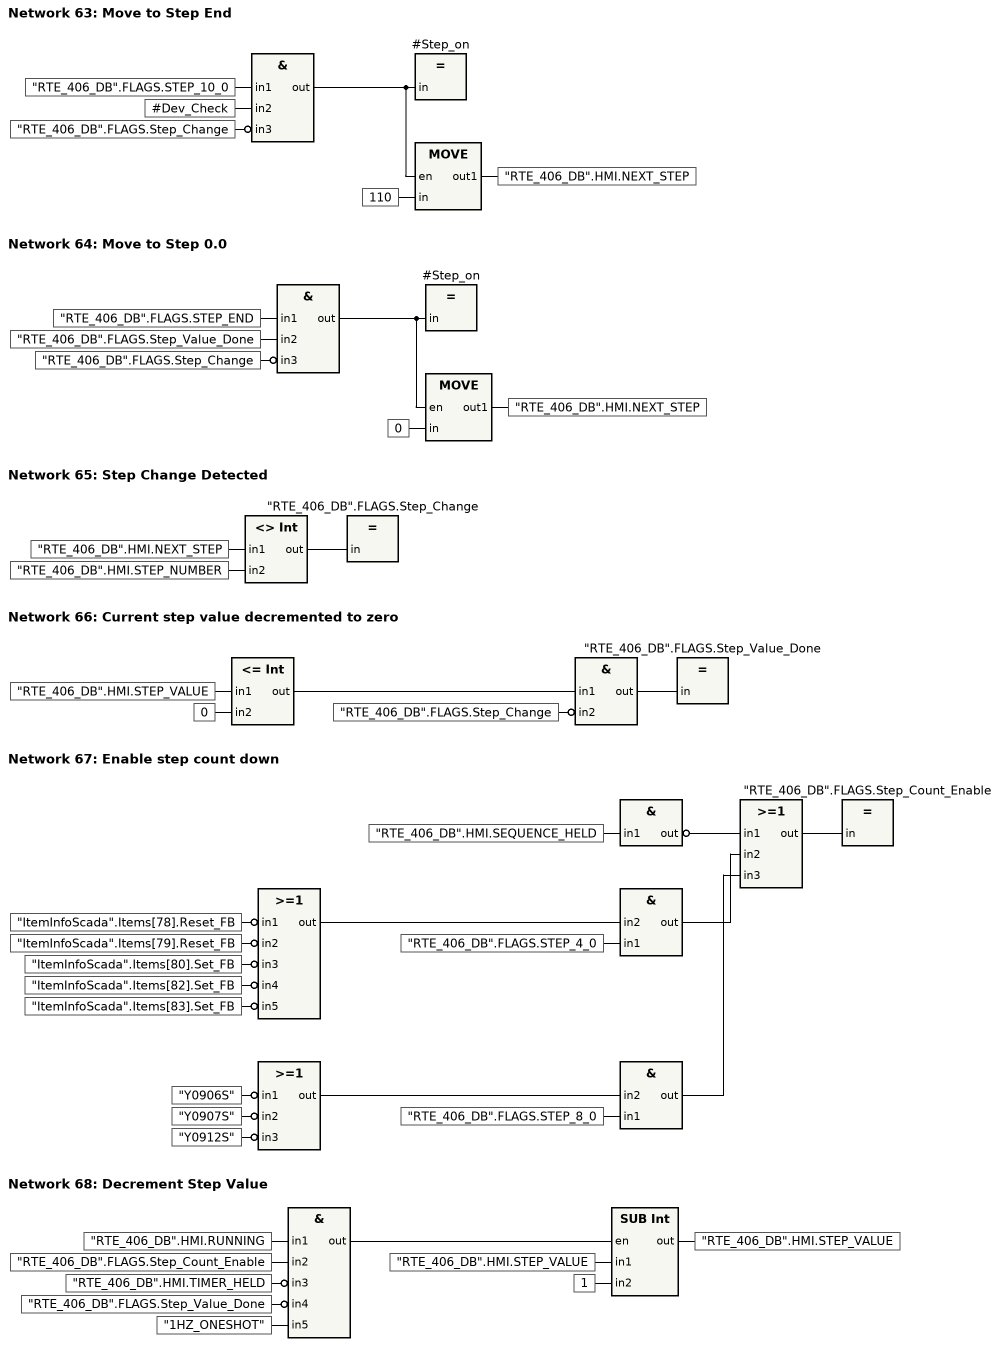
   #Step_on := "RTE_406_DB".FLAGS.STEP_10_0 AND #Dev_Check AND NOT "RTE_406_DB".FLAGS.Step_Change;
   IF #Step_on THEN "RTE_406_DB".HMI.NEXT_STEP := 110; END_IF;
END_REGION

REGION Network 64: Move to Step 0.0
   #Step_on := "RTE_406_DB".FLAGS.STEP_END AND "RTE_406_DB".FLAGS.Step_Value_Done AND NOT "RTE_406_DB".FLAGS.Step_Change;
   IF #Step_on THEN "RTE_406_DB".HMI.NEXT_STEP := 0; END_IF;
END_REGION

REGION Network 65: Step Change Detected
   // The next step number is different to the current step then set flag.
   "RTE_406_DB".FLAGS.Step_Change := "RTE_406_DB".HMI.NEXT_STEP <> "RTE_406_DB".HMI.STEP_NUMBER;
END_REGION

REGION Network 66: Current step value decremented to zero
   "RTE_406_DB".FLAGS.Step_Value_Done := ("RTE_406_DB".HMI.STEP_VALUE <= 0) AND NOT "RTE_406_DB".FLAGS.Step_Change;
END_REGION

REGION Network 67: Enable step count down
   "RTE_406_DB".FLAGS.Step_Count_Enable := NOT "RTE_406_DB".HMI.SEQUENCE_HELD OR ((NOT "ItemInfoScada".Items[78].Reset_FB OR NOT "ItemInfoScada".Items[79].Reset_FB OR NOT "ItemInfoScada".Items[80].Set_FB OR NOT "ItemInfoScada".Items[82].Set_FB OR NOT "ItemInfoScada".Items[83].Set_FB) AND "RTE_406_DB".FLAGS.STEP_4_0) OR ((NOT "Y0906S" OR NOT "Y0907S" OR NOT "Y0912S") AND "RTE_406_DB".FLAGS.STEP_8_0);
END_REGION

REGION Network 68: Decrement Step Value
   // With count enabled and timer not held count down on each 1 second pulse.
   IF "RTE_406_DB".HMI.RUNNING AND "RTE_406_DB".FLAGS.Step_Count_Enable AND NOT "RTE_406_DB".HMI.TIMER_HELD AND NOT "RTE_406_DB".FLAGS.Step_Value_Done AND "1HZ_ONESHOT" THEN
       "RTE_406_DB".HMI.STEP_VALUE := "RTE_406_DB".HMI.STEP_VALUE - 1;
   END_IF;
END_REGION

REGION Network 69: Reset HMI commands
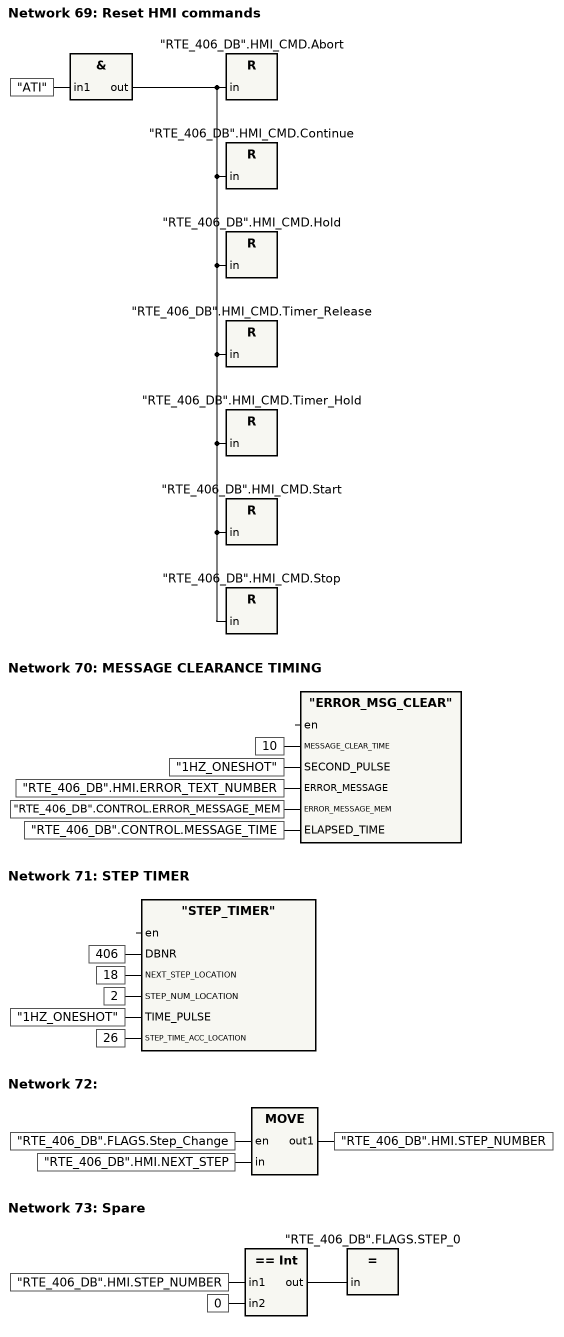
   IF "ATI" THEN
       "RTE_406_DB".HMI_CMD.Abort := FALSE;
       "RTE_406_DB".HMI_CMD.Continue := FALSE;
       "RTE_406_DB".HMI_CMD.Hold := FALSE;
       "RTE_406_DB".HMI_CMD.Timer_Release := FALSE;
       "RTE_406_DB".HMI_CMD.Timer_Hold := FALSE;
       "RTE_406_DB".HMI_CMD.Start := FALSE;
       "RTE_406_DB".HMI_CMD.Stop := FALSE;
   END_IF;
END_REGION

REGION Network 70: MESSAGE CLEARANCE TIMING
   "ERROR_MSG_CLEAR"(MESSAGE_CLEAR_TIME := 10,
                     SECOND_PULSE := "1HZ_ONESHOT",
                     ERROR_MESSAGE := "RTE_406_DB".HMI.ERROR_TEXT_NUMBER,
                     ERROR_MESSAGE_MEM := "RTE_406_DB".CONTROL.ERROR_MESSAGE_MEM,
                     ELAPSED_TIME := "RTE_406_DB".CONTROL.MESSAGE_TIME);
END_REGION

REGION Network 71: STEP TIMER
   // On detection of a new step, the timer is reset to 0 and will then start timing 
   // whilst on the current step.
   "STEP_TIMER"(DBNR := 406,
                NEXT_STEP_LOCATION := 18,
                STEP_NUM_LOCATION := 2,
                TIME_PULSE := "1HZ_ONESHOT",
                STEP_TIME_ACC_LOCATION := 26);
END_REGION

REGION Network 72
   IF "RTE_406_DB".FLAGS.Step_Change THEN "RTE_406_DB".HMI.STEP_NUMBER := "RTE_406_DB".HMI.NEXT_STEP; END_IF;
END_REGION

REGION Network 73: Spare
   "RTE_406_DB".FLAGS.STEP_0 := "RTE_406_DB".HMI.STEP_NUMBER = 0;
END_REGION

REGION Network 74: Spare
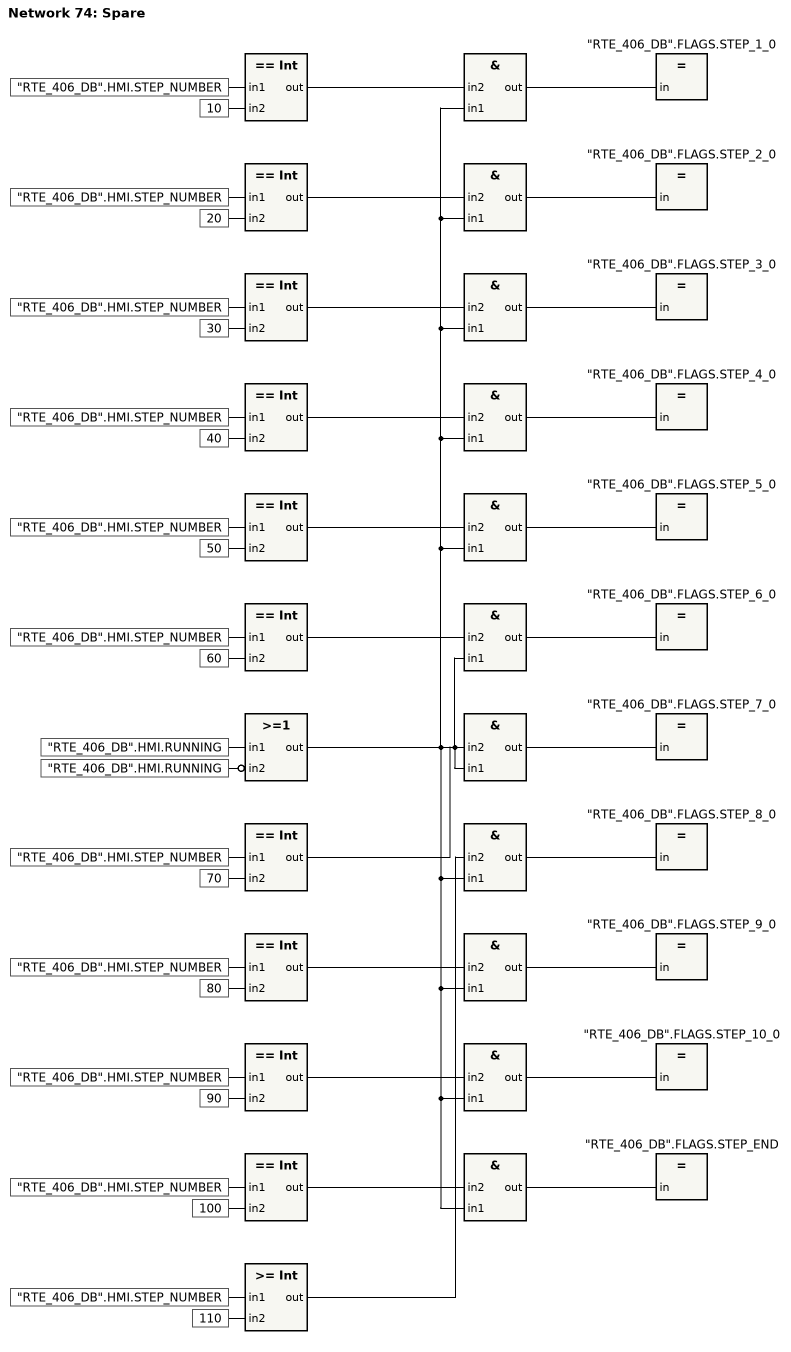
   #_w1 := "RTE_406_DB".HMI.RUNNING OR NOT "RTE_406_DB".HMI.RUNNING;
   "RTE_406_DB".FLAGS.STEP_1_0 := ("RTE_406_DB".HMI.STEP_NUMBER = 10) AND #_w1;
   "RTE_406_DB".FLAGS.STEP_2_0 := ("RTE_406_DB".HMI.STEP_NUMBER = 20) AND #_w1;
   "RTE_406_DB".FLAGS.STEP_3_0 := ("RTE_406_DB".HMI.STEP_NUMBER = 30) AND #_w1;
   "RTE_406_DB".FLAGS.STEP_4_0 := ("RTE_406_DB".HMI.STEP_NUMBER = 40) AND #_w1;
   "RTE_406_DB".FLAGS.STEP_5_0 := ("RTE_406_DB".HMI.STEP_NUMBER = 50) AND #_w1;
   "RTE_406_DB".FLAGS.STEP_6_0 := ("RTE_406_DB".HMI.STEP_NUMBER = 60) AND #_w1;
   "RTE_406_DB".FLAGS.STEP_7_0 := ("RTE_406_DB".HMI.STEP_NUMBER = 70) AND #_w1;
   "RTE_406_DB".FLAGS.STEP_8_0 := ("RTE_406_DB".HMI.STEP_NUMBER = 80) AND #_w1;
   "RTE_406_DB".FLAGS.STEP_9_0 := ("RTE_406_DB".HMI.STEP_NUMBER = 90) AND #_w1;
   "RTE_406_DB".FLAGS.STEP_10_0 := ("RTE_406_DB".HMI.STEP_NUMBER = 100) AND #_w1;
   "RTE_406_DB".FLAGS.STEP_END := ("RTE_406_DB".HMI.STEP_NUMBER >= 110) AND #_w1;
END_REGION

REGION Network 75: COPY CURRENT STEP TO STEP TEXT WORD
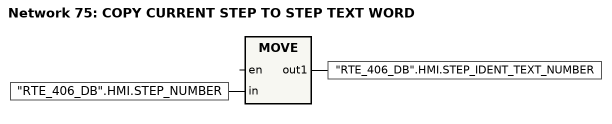
   "RTE_406_DB".HMI.STEP_IDENT_TEXT_NUMBER := "RTE_406_DB".HMI.STEP_NUMBER;
END_REGION
END_FUNCTION
